// TIA Portal V19 export
FUNCTION_BLOCK "LiftSim"   // FB14, FBD
TITLE = LiftSim
{ S7_Optimized_Access := 'TRUE' }
AUTHOR : Siemens
// Simulation BeltLift
// stored: IsIECCheckEnabled true, MemoryReserve 100, SetENOAutomatically true
   VAR
      instRisTrigLift1 { ExternalAccessible := 'False'; ExternalVisible := 'False'; ExternalWritable := 'False'; S7_SetPoint := 'True'} : R_TRIG;
      instRisTrigLift2 { ExternalAccessible := 'False'; ExternalVisible := 'False'; ExternalWritable := 'False'; S7_SetPoint := 'True'} : R_TRIG;
      statRisTrigLift1 { ExternalAccessible := 'False'; ExternalVisible := 'False'; ExternalWritable := 'False'} : Bool;
      statRisTrigLift2 { ExternalAccessible := 'False'; ExternalVisible := 'False'; ExternalWritable := 'False'} : Bool;
      instRisTrigClock { ExternalAccessible := 'False'; ExternalVisible := 'False'; ExternalWritable := 'False'; S7_SetPoint := 'True'} : R_TRIG;
      statRisTrigClock { ExternalAccessible := 'False'; ExternalVisible := 'False'; ExternalWritable := 'False'} : Bool;
      statClock10Hz { ExternalAccessible := 'False'; ExternalVisible := 'False'; ExternalWritable := 'False'} : Bool;
      instMovingLightBelt { ExternalAccessible := 'False'; ExternalVisible := 'False'; ExternalWritable := 'False'; S7_SetPoint := 'True'} : "MovingLight";
      instMovingLightLift1 { ExternalAccessible := 'False'; ExternalVisible := 'False'; ExternalWritable := 'False'; S7_SetPoint := 'True'} : "MovingLight";
      instMovingLightLift2 { ExternalAccessible := 'False'; ExternalVisible := 'False'; ExternalWritable := 'False'; S7_SetPoint := 'True'} : "MovingLight";
      statDirBelt { ExternalAccessible := 'False'; ExternalVisible := 'False'; ExternalWritable := 'False'} : Int;
      statDirLift1 { ExternalAccessible := 'False'; ExternalVisible := 'False'; ExternalWritable := 'False'} : Int;
      statDirLift2 { ExternalAccessible := 'False'; ExternalVisible := 'False'; ExternalWritable := 'False'} : Int;
      instLEDsBelt { ExternalAccessible := 'False'; ExternalVisible := 'False'; ExternalWritable := 'False'; S7_SetPoint := 'True'} : "LEDs";
      instLEDsLift1 { ExternalAccessible := 'False'; ExternalVisible := 'False'; ExternalWritable := 'False'; S7_SetPoint := 'True'} : "LEDs";
      instLEDsLift2 { ExternalAccessible := 'False'; ExternalVisible := 'False'; ExternalWritable := 'False'; S7_SetPoint := 'True'} : "LEDs";
   END_VAR
BEGIN

REGION Network 1
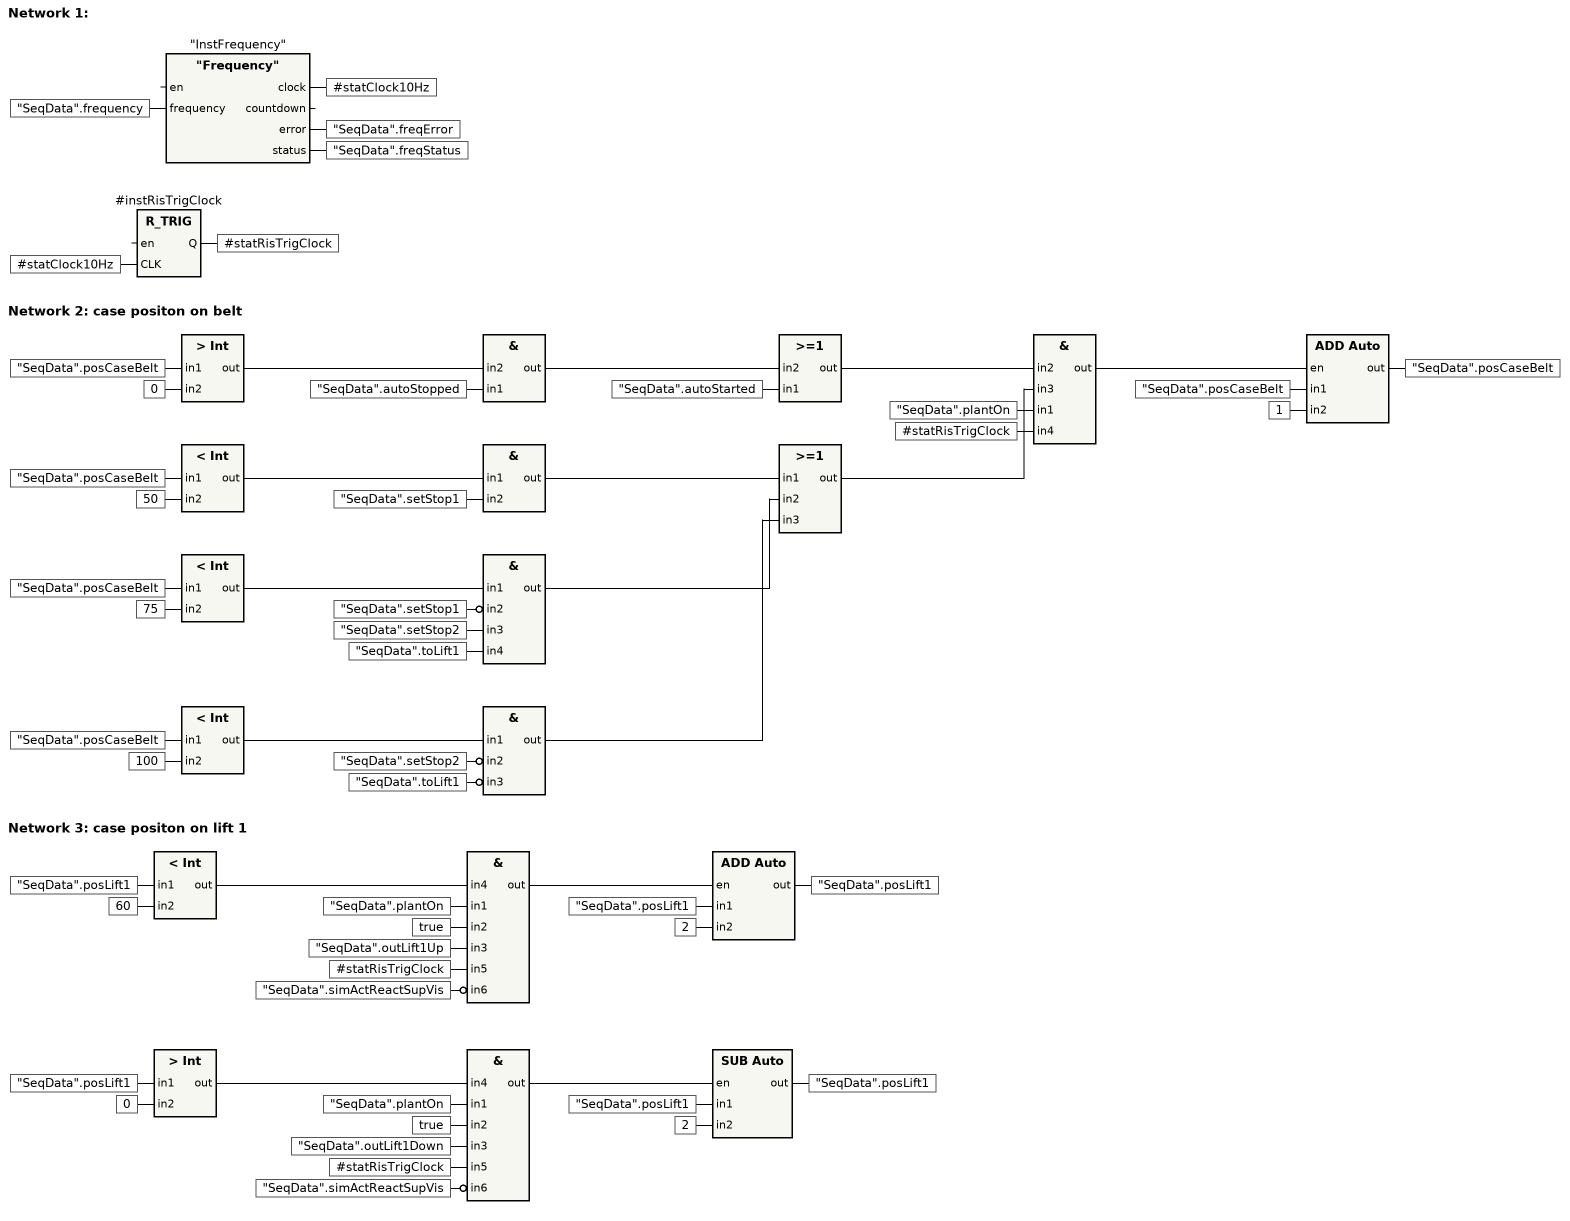
   "InstFrequency"(frequency := "SeqData".frequency,   // "Frequency"
                   clock => #statClock10Hz,
                   error => "SeqData".freqError,
                   status => "SeqData".freqStatus);
   #instRisTrigClock(CLK := #statClock10Hz, Q => #statRisTrigClock);   // R_TRIG
END_REGION

REGION Network 2: case positon on belt
   IF ((("SeqData".posCaseBelt > 0) AND "SeqData".autoStopped) OR "SeqData".autoStarted) AND ((("SeqData".posCaseBelt < 50) AND "SeqData".setStop1) OR (("SeqData".posCaseBelt < 75) AND NOT "SeqData".setStop1 AND "SeqData".setStop2 AND "SeqData".toLift1) OR (("SeqData".posCaseBelt < 100) AND NOT "SeqData".setStop2 AND NOT "SeqData".toLift1)) AND "SeqData".plantOn AND #statRisTrigClock THEN
       "SeqData".posCaseBelt := "SeqData".posCaseBelt + 1;
   END_IF;
END_REGION

REGION Network 3: case positon on lift 1
   IF ("SeqData".posLift1 < 60) AND "SeqData".plantOn AND true AND "SeqData".outLift1Up AND #statRisTrigClock AND NOT "SeqData".simActReactSupVis THEN
       "SeqData".posLift1 := "SeqData".posLift1 + 2;
   END_IF;
   IF ("SeqData".posLift1 > 0) AND "SeqData".plantOn AND true AND "SeqData".outLift1Down AND #statRisTrigClock AND NOT "SeqData".simActReactSupVis THEN
       "SeqData".posLift1 := "SeqData".posLift1 - 2;
   END_IF;
END_REGION

REGION Network 4: case positon on lift 2
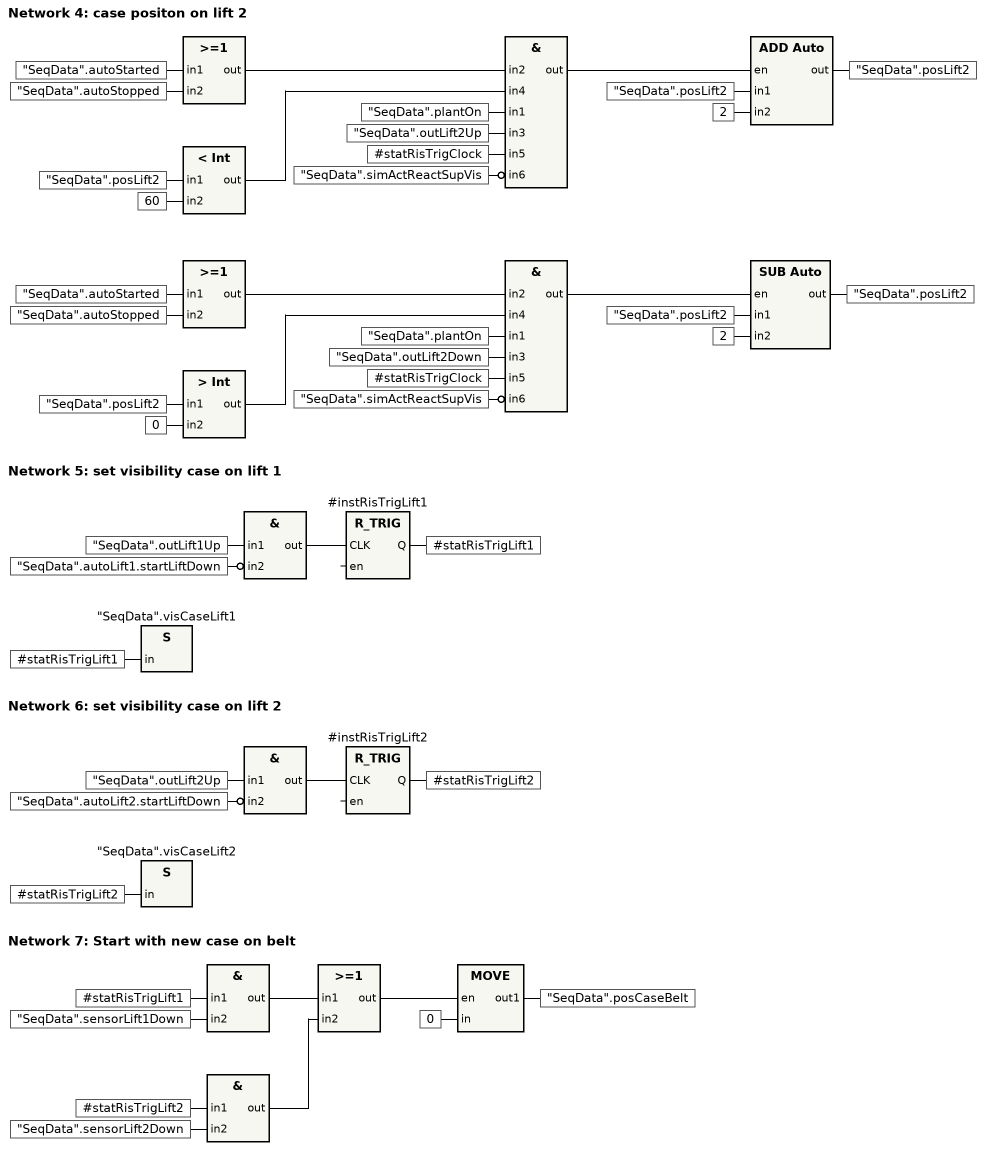
   IF ("SeqData".autoStarted OR "SeqData".autoStopped) AND ("SeqData".posLift2 < 60) AND "SeqData".plantOn AND "SeqData".outLift2Up AND #statRisTrigClock AND NOT "SeqData".simActReactSupVis THEN
       "SeqData".posLift2 := "SeqData".posLift2 + 2;
   END_IF;
   IF ("SeqData".autoStarted OR "SeqData".autoStopped) AND ("SeqData".posLift2 > 0) AND "SeqData".plantOn AND "SeqData".outLift2Down AND #statRisTrigClock AND NOT "SeqData".simActReactSupVis THEN
       "SeqData".posLift2 := "SeqData".posLift2 - 2;
   END_IF;
END_REGION

REGION Network 5: set visibility case on lift 1
   #instRisTrigLift1(CLK := "SeqData".outLift1Up AND NOT "SeqData".autoLift1.startLiftDown,   // R_TRIG
                     Q => #statRisTrigLift1);
   IF #statRisTrigLift1 THEN "SeqData".visCaseLift1 := TRUE; END_IF;
END_REGION

REGION Network 6: set visibility case on lift 2
   #instRisTrigLift2(CLK := "SeqData".outLift2Up AND NOT "SeqData".autoLift2.startLiftDown,   // R_TRIG
                     Q => #statRisTrigLift2);
   IF #statRisTrigLift2 THEN "SeqData".visCaseLift2 := TRUE; END_IF;
END_REGION

REGION Network 7: Start with new case on belt
   IF (#statRisTrigLift1 AND "SeqData".sensorLift1Down) OR (#statRisTrigLift2 AND "SeqData".sensorLift2Down) THEN
       "SeqData".posCaseBelt := 0;
   END_IF;
END_REGION

REGION Network 8: check, if new case
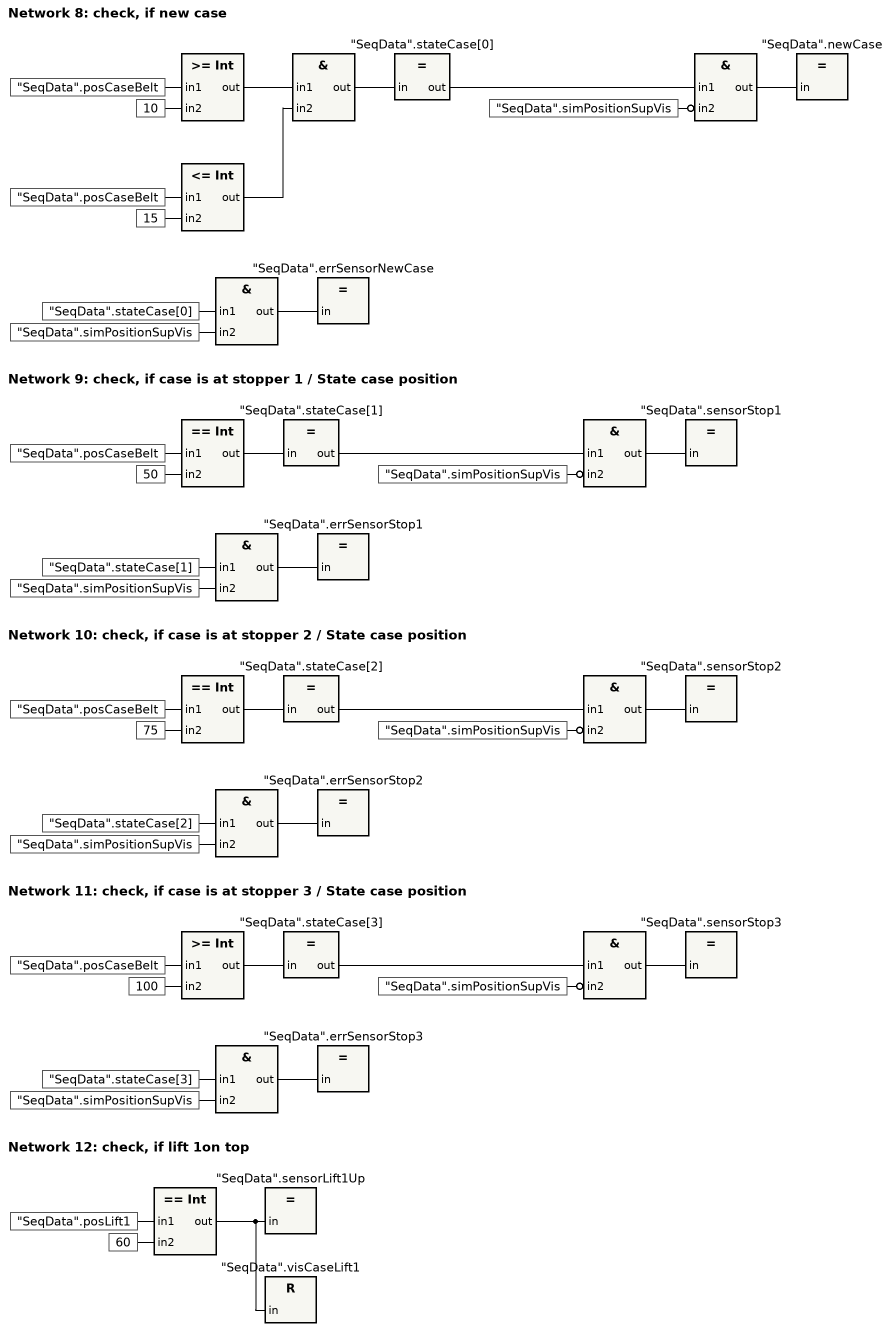
   "SeqData".stateCase[0] := ("SeqData".posCaseBelt >= 10) AND ("SeqData".posCaseBelt <= 15);
   "SeqData".newCase := ("SeqData".posCaseBelt >= 10) AND ("SeqData".posCaseBelt <= 15) AND NOT "SeqData".simPositionSupVis;
   "SeqData".errSensorNewCase := "SeqData".stateCase[0] AND "SeqData".simPositionSupVis;
END_REGION

REGION Network 9: check, if case is at stopper 1 / State case position
   "SeqData".stateCase[1] := "SeqData".posCaseBelt = 50;
   "SeqData".sensorStop1 := ("SeqData".posCaseBelt = 50) AND NOT "SeqData".simPositionSupVis;
   "SeqData".errSensorStop1 := "SeqData".stateCase[1] AND "SeqData".simPositionSupVis;
END_REGION

REGION Network 10: check, if case is at stopper 2 / State case position
   "SeqData".stateCase[2] := "SeqData".posCaseBelt = 75;
   "SeqData".sensorStop2 := ("SeqData".posCaseBelt = 75) AND NOT "SeqData".simPositionSupVis;
   "SeqData".errSensorStop2 := "SeqData".stateCase[2] AND "SeqData".simPositionSupVis;
END_REGION

REGION Network 11: check, if case is at stopper 3 / State case position
   "SeqData".stateCase[3] := "SeqData".posCaseBelt >= 100;
   "SeqData".sensorStop3 := ("SeqData".posCaseBelt >= 100) AND NOT "SeqData".simPositionSupVis;
   "SeqData".errSensorStop3 := "SeqData".stateCase[3] AND "SeqData".simPositionSupVis;
END_REGION

REGION Network 12: check, if lift 1on top
   "SeqData".sensorLift1Up := "SeqData".posLift1 = 60;
   IF "SeqData".sensorLift1Up THEN "SeqData".visCaseLift1 := FALSE; END_IF;
END_REGION

REGION Network 13: check, if lift 2 on top
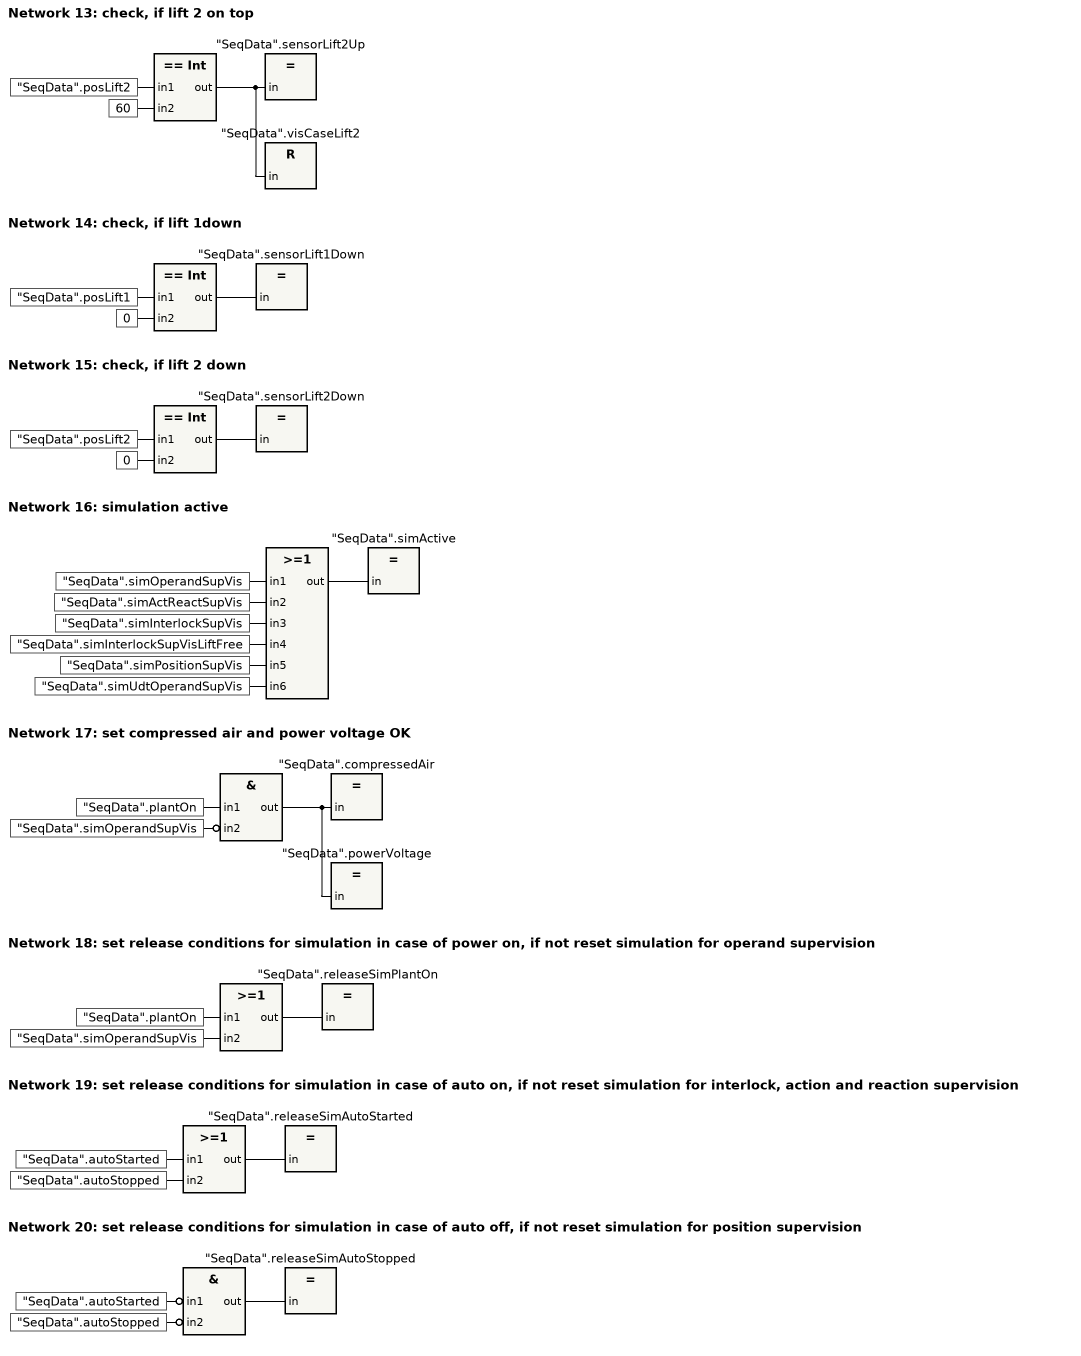
   "SeqData".sensorLift2Up := "SeqData".posLift2 = 60;
   IF "SeqData".sensorLift2Up THEN "SeqData".visCaseLift2 := FALSE; END_IF;
END_REGION

REGION Network 14: check, if lift 1down
   "SeqData".sensorLift1Down := "SeqData".posLift1 = 0;
END_REGION

REGION Network 15: check, if lift 2 down
   "SeqData".sensorLift2Down := "SeqData".posLift2 = 0;
END_REGION

REGION Network 16: simulation active
   "SeqData".simActive := "SeqData".simOperandSupVis OR "SeqData".simActReactSupVis OR "SeqData".simInterlockSupVis OR "SeqData".simInterlockSupVisLiftFree OR "SeqData".simPositionSupVis OR "SeqData".simUdtOperandSupVis;
END_REGION

REGION Network 17: set compressed air and power voltage OK
   "SeqData".compressedAir := "SeqData".plantOn AND NOT "SeqData".simOperandSupVis;
   "SeqData".powerVoltage := "SeqData".compressedAir;
END_REGION

REGION Network 18: set release conditions for simulation in case of power on, if not reset simulation for operand supervision
   "SeqData".releaseSimPlantOn := "SeqData".plantOn OR "SeqData".simOperandSupVis;
END_REGION

REGION Network 19: set release conditions for simulation in case of auto on, if not reset simulation for interlock, action and reaction supervision
   "SeqData".releaseSimAutoStarted := "SeqData".autoStarted OR "SeqData".autoStopped;
END_REGION

REGION Network 20: set release conditions for simulation in case of auto off, if not reset simulation for position supervision
   "SeqData".releaseSimAutoStopped := NOT "SeqData".autoStarted AND NOT "SeqData".autoStopped;
END_REGION

REGION Network 21: set door closed
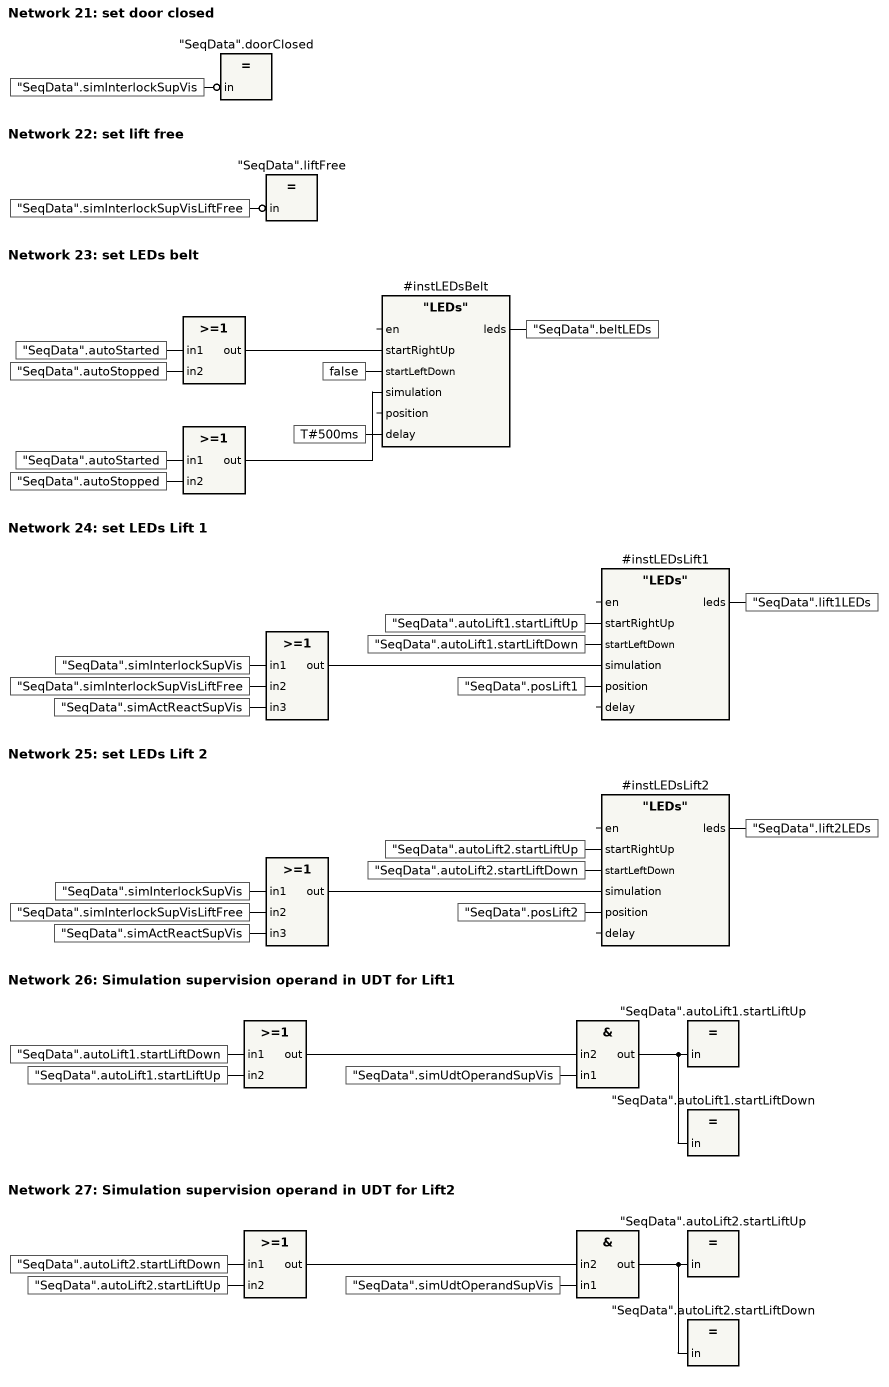
   "SeqData".doorClosed := NOT "SeqData".simInterlockSupVis;
END_REGION

REGION Network 22: set lift free
   "SeqData".liftFree := NOT "SeqData".simInterlockSupVisLiftFree;
END_REGION

REGION Network 23: set LEDs belt
   #instLEDsBelt(startRightUp := "SeqData".autoStarted OR "SeqData".autoStopped,   // "LEDs"
                 startLeftDown := false,
                 simulation := "SeqData".autoStarted OR "SeqData".autoStopped,
                 delay := T#500ms,
                 leds => "SeqData".beltLEDs);
END_REGION

REGION Network 24: set LEDs Lift 1
   #instLEDsLift1(startRightUp := "SeqData".autoLift1.startLiftUp,   // "LEDs"
                  startLeftDown := "SeqData".autoLift1.startLiftDown,
                  simulation := "SeqData".simInterlockSupVis OR "SeqData".simInterlockSupVisLiftFree OR "SeqData".simActReactSupVis,
                  position := "SeqData".posLift1,
                  leds => "SeqData".lift1LEDs);
END_REGION

REGION Network 25: set LEDs Lift 2
   #instLEDsLift2(startRightUp := "SeqData".autoLift2.startLiftUp,   // "LEDs"
                  startLeftDown := "SeqData".autoLift2.startLiftDown,
                  simulation := "SeqData".simInterlockSupVis OR "SeqData".simInterlockSupVisLiftFree OR "SeqData".simActReactSupVis,
                  position := "SeqData".posLift2,
                  leds => "SeqData".lift2LEDs);
END_REGION

REGION Network 26: Simulation supervision operand in UDT for Lift1
   "SeqData".autoLift1.startLiftUp := ("SeqData".autoLift1.startLiftDown OR "SeqData".autoLift1.startLiftUp) AND "SeqData".simUdtOperandSupVis;
   "SeqData".autoLift1.startLiftDown := "SeqData".autoLift1.startLiftUp;
END_REGION

REGION Network 27: Simulation supervision operand in UDT for Lift2
   "SeqData".autoLift2.startLiftUp := ("SeqData".autoLift2.startLiftDown OR "SeqData".autoLift2.startLiftUp) AND "SeqData".simUdtOperandSupVis;
   "SeqData".autoLift2.startLiftDown := "SeqData".autoLift2.startLiftUp;
END_REGION
END_FUNCTION_BLOCK
